PROGRAM LadderLogic
VAR
	MC_Halt_0: MC_Halt;
END_VAR

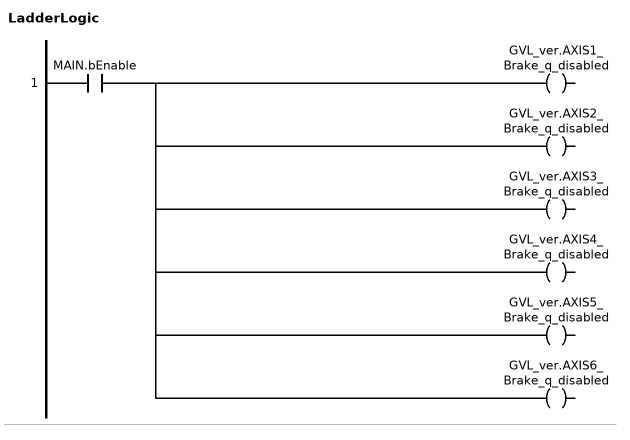
// NETWORK 1
GVL_ver.AXIS1_Brake_q_disabled := MAIN.bEnable;
GVL_ver.AXIS2_Brake_q_disabled := MAIN.bEnable;
GVL_ver.AXIS3_Brake_q_disabled := MAIN.bEnable;
GVL_ver.AXIS4_Brake_q_disabled := MAIN.bEnable;
GVL_ver.AXIS5_Brake_q_disabled := MAIN.bEnable;
GVL_ver.AXIS6_Brake_q_disabled := MAIN.bEnable;

END_PROGRAM

(* stored: Version 1.1.0.1, ProductVersion 3.1.4022.3
   POU LadderLogic: Id {b2a6c3af-5afe-4924-a72e-c164c2aa7008}, SpecialFunc None *)
